// TIA Portal V21 export
FUNCTION "VACCUM" : Void   // FC12, LAD
{ S7_Optimized_Access := 'TRUE' }
// stored: SetENOAutomatically false
   VAR_TEMP
      "VACCUM DIFF" : Real;
      "VACCUM LEAK DIFF" : Real;
   END_VAR
   VAR_TEMP   // added for the SCL form of the ladder/FBD networks
      _w1 : Bool;
      _w2 : Bool;
      _w3 : Bool;
      _w4 : Bool;
      _w5 : Bool;
      _w6 : Bool;
      _w7 : Bool;
      _w8 : Bool;
      _w9 : Bool;
      _w10 : Bool;
      _w11 : Bool;
      _w12 : Bool;
      _w13 : Bool;
      _w14 : Bool;
      _w15 : Bool;
      _w16 : Bool;
      _w17 : Bool;
      _w18 : Bool;
      _w19 : Bool;
      _w20 : Bool;
   END_VAR
BEGIN

REGION Network 1
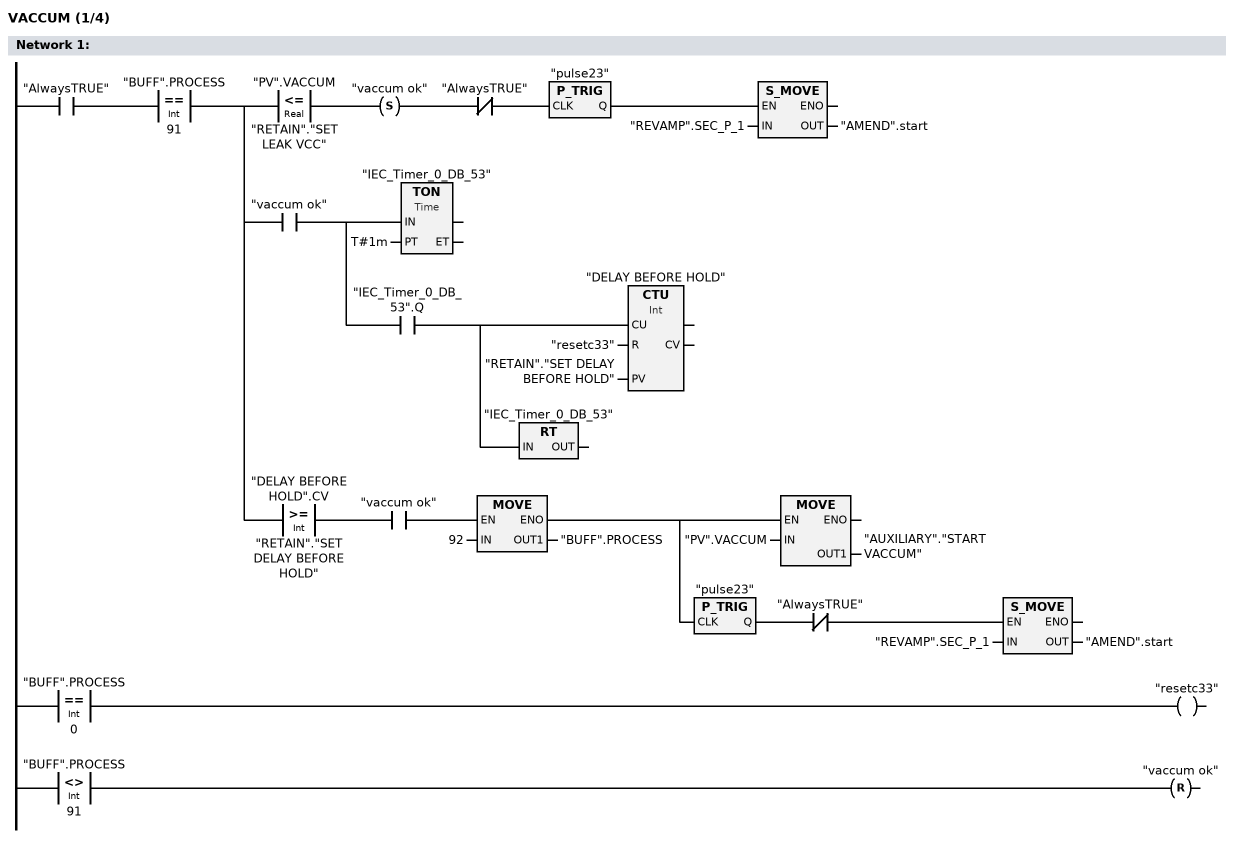
   RUNG wire#powerrail
      Contact( "AlwaysTRUE" )
      { S7_Templates := "SrcType := Int" } EQ_Contact(in1 := "BUFF".PROCESS, in2 := 91)
      wire#w1
      { S7_Templates := "SrcType := Real" } LE_Contact(in1 := "PV".VACCUM, in2 := "RETAIN"."SET LEAK VCC")
      S_Coil( "vaccum ok" )
      I_Contact( "AlwaysTRUE" )
      P_Trig( "pulse23" )
      S_Move(in := "REVAMP".SEC_P_1, out => "AMEND".start)
   END_RUNG
   RUNG wire#w1
      Contact( "vaccum ok" )
      wire#w2
      { S7_Templates := "time_type := Time" } "IEC_Timer_0_DB_53".TON(pt := T#1m, et =>)
   END_RUNG
   RUNG wire#w2
      Contact( "IEC_Timer_0_DB_53".Q )
      wire#w3
      { S7_Templates := "value_type := Int" } "DELAY BEFORE HOLD".CTU(r := "resetc33", pv := "RETAIN"."SET DELAY BEFORE HOLD", cv =>)
   END_RUNG
   RUNG wire#w3
      RT_Coil( "IEC_Timer_0_DB_53" )
   END_RUNG
   RUNG wire#w1
      { S7_Templates := "SrcType := Int" } GE_Contact(in1 := "DELAY BEFORE HOLD".CV, in2 := "RETAIN"."SET DELAY BEFORE HOLD")
      Contact( "vaccum ok" )
      Move(in := 92, out1 => "BUFF".PROCESS)
      wire#w4
      Move(in := "PV".VACCUM, out1 => "AUXILIARY"."START VACCUM")
   END_RUNG
   RUNG wire#w4
      P_Trig( "pulse23" )
      I_Contact( "AlwaysTRUE" )
      S_Move(in := "REVAMP".SEC_P_1, out => "AMEND".start)
   END_RUNG
   RUNG wire#powerrail
      { S7_Templates := "SrcType := Int" } EQ_Contact(in1 := "BUFF".PROCESS, in2 := 0)
      Coil( "resetc33" )
   END_RUNG
   RUNG wire#powerrail
      { S7_Templates := "SrcType := Int" } NE_Contact(in1 := "BUFF".PROCESS, in2 := 91)
      R_Coil( "vaccum ok" )
   END_RUNG
   // the same network as SCL:
   #_w1 := "AlwaysTRUE" AND ("BUFF".PROCESS = 91);
   #_w2 := #_w1 AND ("PV".VACCUM <= "RETAIN"."SET LEAK VCC");
   IF #_w2 THEN "vaccum ok" := TRUE; END_IF;
   #_w3 := #_w2 AND NOT "AlwaysTRUE";
   #_w4 := #_w3 AND NOT "pulse23";   // rising edge
   "pulse23" := #_w3;
   IF #_w4 THEN "AMEND".start := "REVAMP".SEC_P_1; END_IF;
   #_w5 := #_w1 AND "vaccum ok";
   "IEC_Timer_0_DB_53".TON(IN := #_w5, PT := T#1m);
   #_w6 := #_w5 AND "IEC_Timer_0_DB_53".Q;
   "DELAY BEFORE HOLD".CTU(CU := #_w6, R := "resetc33", PV := "RETAIN"."SET DELAY BEFORE HOLD");
   IF #_w6 THEN RESET_TIMER("IEC_Timer_0_DB_53"); END_IF;
   #_w7 := #_w1 AND ("DELAY BEFORE HOLD".CV >= "RETAIN"."SET DELAY BEFORE HOLD") AND "vaccum ok";
   IF #_w7 THEN
       "BUFF".PROCESS := 92;
       "AUXILIARY"."START VACCUM" := "PV".VACCUM;
   END_IF;
   #_w8 := #_w7 AND NOT "pulse23";   // rising edge
   "pulse23" := #_w7;
   IF #_w8 AND NOT "AlwaysTRUE" THEN "AMEND".start := "REVAMP".SEC_P_1; END_IF;
   "resetc33" := "BUFF".PROCESS = 0;
   IF "BUFF".PROCESS <> 91 THEN "vaccum ok" := FALSE; END_IF;
END_REGION

REGION Network 2
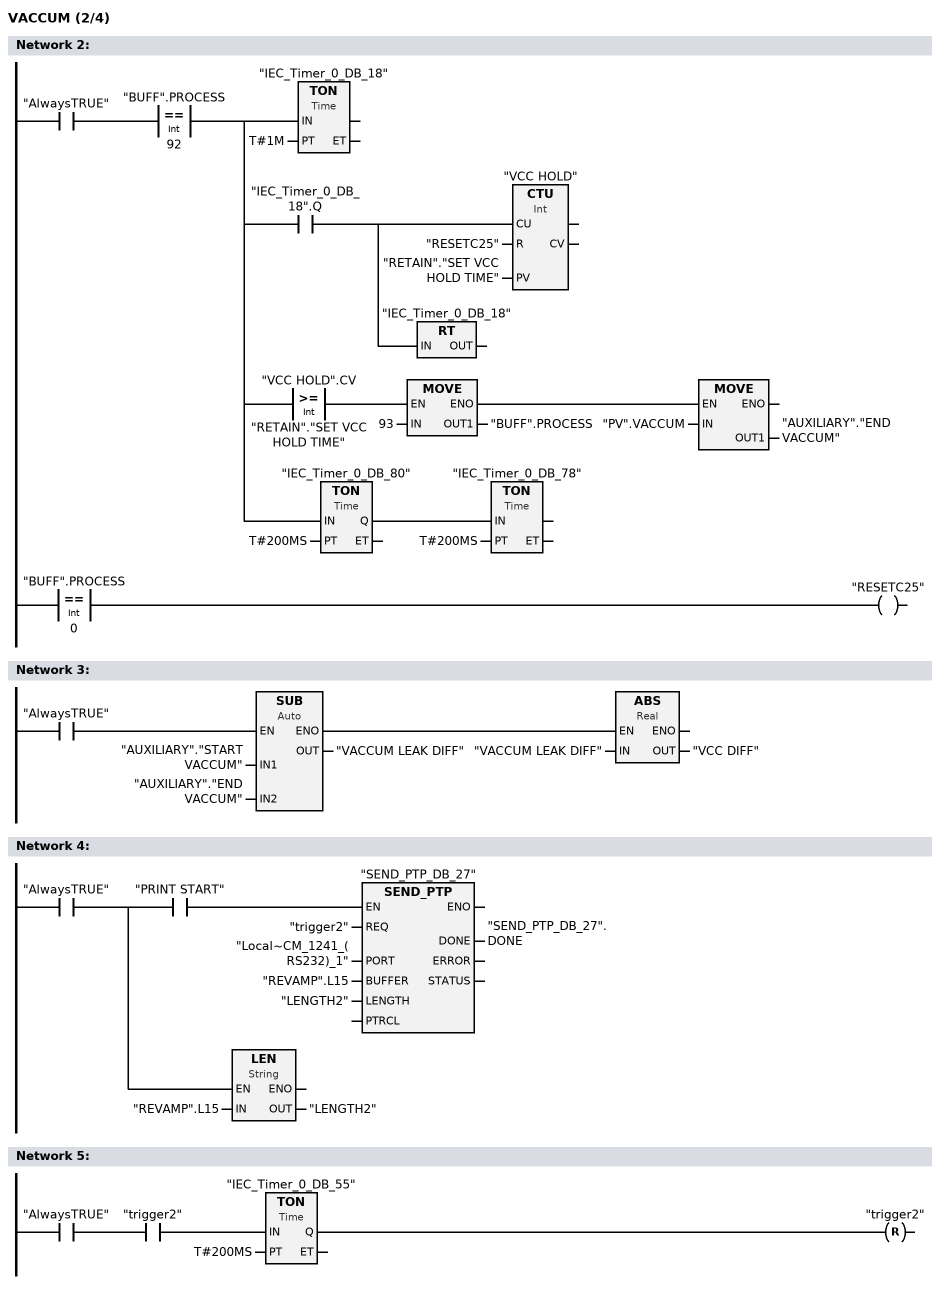
   RUNG wire#powerrail
      Contact( "AlwaysTRUE" )
      { S7_Templates := "SrcType := Int" } EQ_Contact(in1 := "BUFF".PROCESS, in2 := 92)
      wire#w1
      { S7_Templates := "time_type := Time" } "IEC_Timer_0_DB_18".TON(pt := T#1M, et =>)
   END_RUNG
   RUNG wire#w1
      Contact( "IEC_Timer_0_DB_18".Q )
      wire#w2
      { S7_Templates := "value_type := Int" } "VCC HOLD".CTU(r := "RESETC25", pv := "RETAIN"."SET VCC HOLD TIME", cv =>)
   END_RUNG
   RUNG wire#w2
      RT_Coil( "IEC_Timer_0_DB_18" )
   END_RUNG
   RUNG wire#w1
      { S7_Templates := "SrcType := Int" } GE_Contact(in1 := "VCC HOLD".CV, in2 := "RETAIN"."SET VCC HOLD TIME")
      Move(in := 93, out1 => "BUFF".PROCESS)
      Move(in := "PV".VACCUM, out1 => "AUXILIARY"."END VACCUM")
   END_RUNG
   RUNG wire#w1
      { S7_Templates := "time_type := Time" } "IEC_Timer_0_DB_80".TON(pt := T#200MS, et =>)
      { S7_Templates := "time_type := Time" } "IEC_Timer_0_DB_78".TON(pt := T#200MS, et =>)
   END_RUNG
   RUNG wire#powerrail
      { S7_Templates := "SrcType := Int" } EQ_Contact(in1 := "BUFF".PROCESS, in2 := 0)
      Coil( "RESETC25" )
   END_RUNG
   // the same network as SCL:
   #_w1 := "AlwaysTRUE" AND ("BUFF".PROCESS = 92);
   "IEC_Timer_0_DB_18".TON(IN := #_w1, PT := T#1M);
   #_w2 := #_w1 AND "IEC_Timer_0_DB_18".Q;
   "VCC HOLD".CTU(CU := #_w2, R := "RESETC25", PV := "RETAIN"."SET VCC HOLD TIME");
   IF #_w2 THEN RESET_TIMER("IEC_Timer_0_DB_18"); END_IF;
   IF #_w1 AND ("VCC HOLD".CV >= "RETAIN"."SET VCC HOLD TIME") THEN
       "BUFF".PROCESS := 93;
       "AUXILIARY"."END VACCUM" := "PV".VACCUM;
   END_IF;
   "IEC_Timer_0_DB_80".TON(IN := #_w1, PT := T#200MS);
   "IEC_Timer_0_DB_78".TON(IN := "IEC_Timer_0_DB_80".Q, PT := T#200MS);
   "RESETC25" := "BUFF".PROCESS = 0;
END_REGION

REGION Network 3
   RUNG wire#powerrail
      Contact( "AlwaysTRUE" )
      Sub(in1 := "AUXILIARY"."START VACCUM", in2 := "AUXILIARY"."END VACCUM", out => "VACCUM LEAK DIFF")
      { S7_Templates := "SrcType := Real" } Abs(in := "VACCUM LEAK DIFF", out => "VCC DIFF")
   END_RUNG
   // the same network as SCL:
   IF "AlwaysTRUE" THEN
       "VACCUM LEAK DIFF" := "AUXILIARY"."START VACCUM" - "AUXILIARY"."END VACCUM";
       "VCC DIFF" := ABS("VACCUM LEAK DIFF");
   END_IF;
END_REGION

REGION Network 4
   RUNG wire#powerrail
      Contact( "AlwaysTRUE" )
      wire#w1
      Contact( "PRINT START" )
      "SEND_PTP_DB_27".SEND_PTP(REQ := "trigger2", PORT := "Local~CM_1241_(RS232)_1", BUFFER := "REVAMP".L15, LENGTH := "LENGTH2", PTRCL :=, DONE => "SEND_PTP_DB_27".DONE, ERROR =>, STATUS =>)
   END_RUNG
   RUNG wire#w1
      { S7_Templates := "[str_type := String, return_type := Int]" } LEN(IN := "REVAMP".L15, OUT => "LENGTH2")
   END_RUNG
   // the same network as SCL:
   #_w1 := "AlwaysTRUE";
   IF "AlwaysTRUE" AND "PRINT START" THEN
       "SEND_PTP_DB_27"(REQ := "trigger2",   // SEND_PTP
                        PORT := "Local~CM_1241_(RS232)_1",
                        BUFFER := "REVAMP".L15,
                        LENGTH := "LENGTH2",
                        DONE => "SEND_PTP_DB_27".DONE);
   END_IF;
   IF #_w1 THEN LEN(IN := "REVAMP".L15, OUT => "LENGTH2"); END_IF;
END_REGION

REGION Network 5
   RUNG wire#powerrail
      Contact( "AlwaysTRUE" )
      Contact( "trigger2" )
      { S7_Templates := "time_type := Time" } "IEC_Timer_0_DB_55".TON(pt := T#200MS, et =>)
      R_Coil( "trigger2" )
   END_RUNG
   // the same network as SCL:
   "IEC_Timer_0_DB_55".TON(IN := "AlwaysTRUE" AND "trigger2", PT := T#200MS);
   IF "IEC_Timer_0_DB_55".Q THEN "trigger2" := FALSE; END_IF;
END_REGION

REGION Network 6
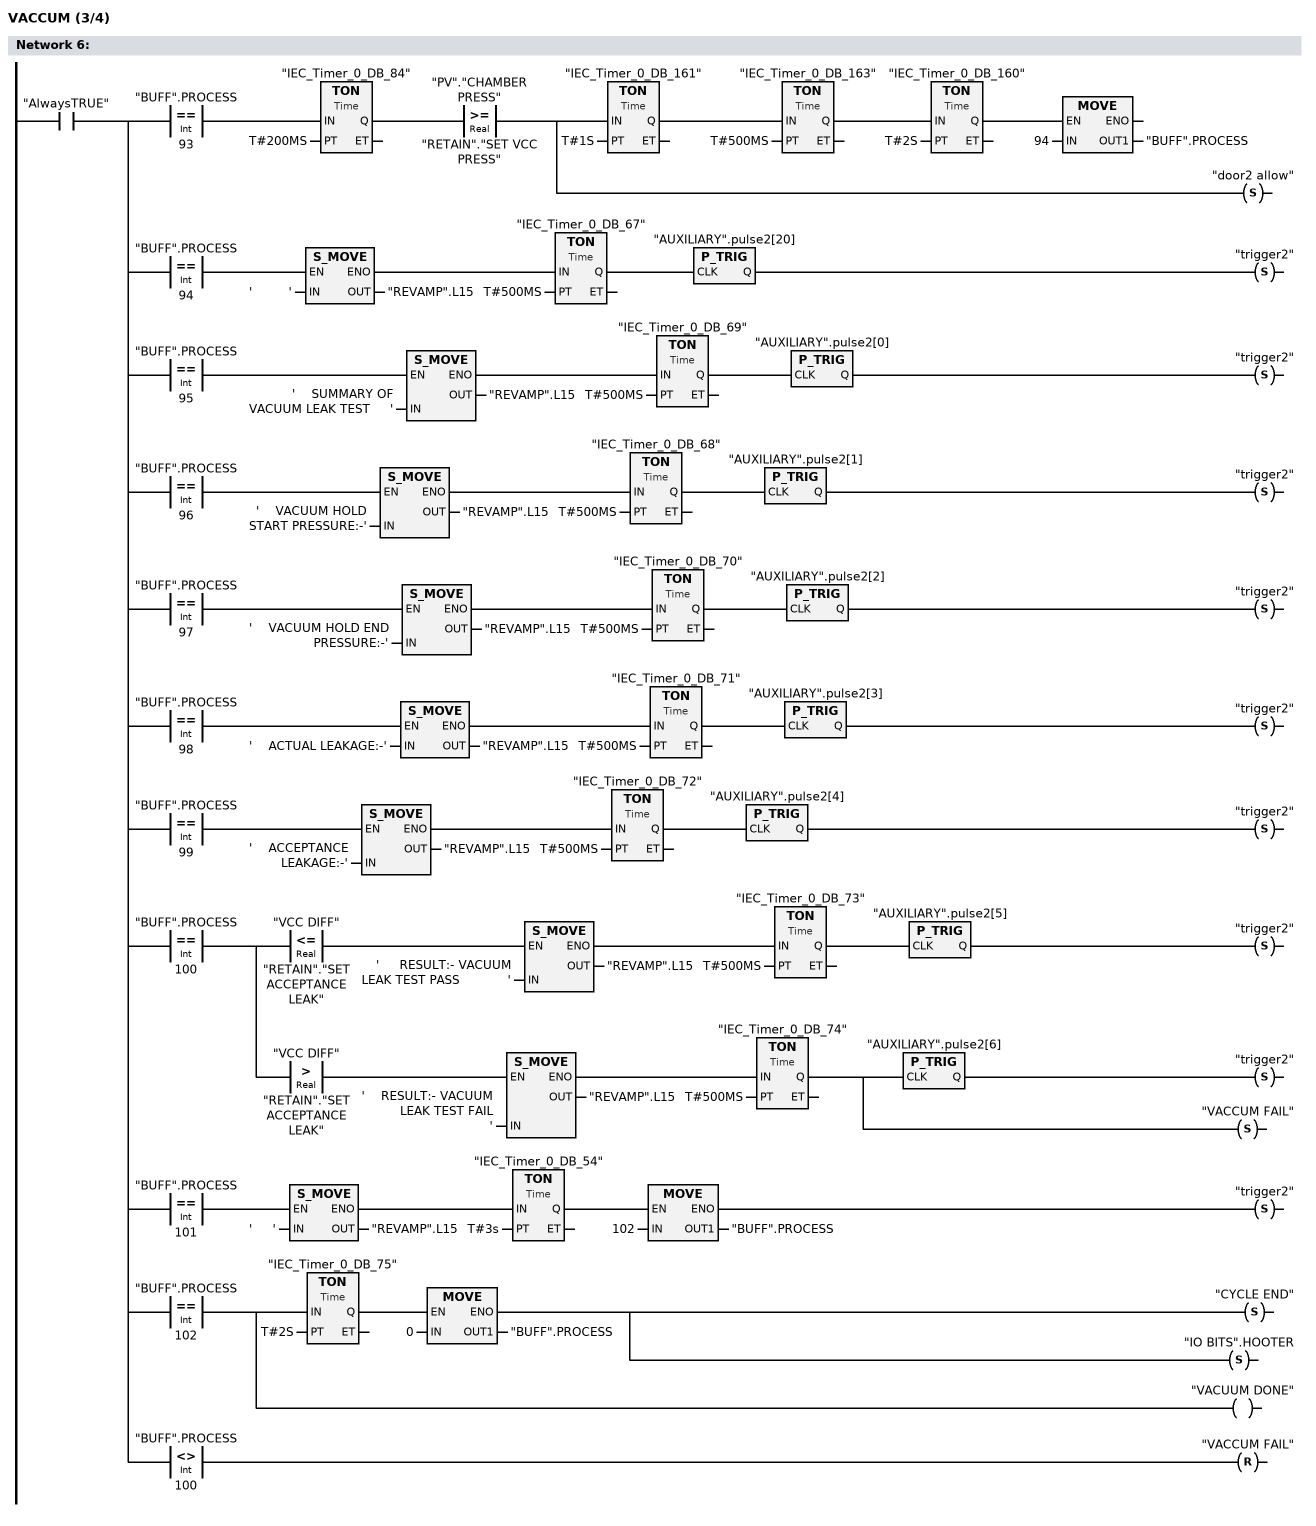
   RUNG wire#powerrail
      Contact( "AlwaysTRUE" )
      wire#w1
      { S7_Templates := "SrcType := Int" } EQ_Contact(in1 := "BUFF".PROCESS, in2 := 93)
      { S7_Templates := "time_type := Time" } "IEC_Timer_0_DB_84".TON(pt := T#200MS, et =>)
      { S7_Templates := "SrcType := Real" } GE_Contact(in1 := "PV"."CHAMBER PRESS", in2 := "RETAIN"."SET VCC PRESS")
      wire#w2
      { S7_Templates := "time_type := Time" } "IEC_Timer_0_DB_161".TON(pt := T#1S, et =>)
      { S7_Templates := "time_type := Time" } "IEC_Timer_0_DB_163".TON(pt := T#500MS, et =>)
      { S7_Templates := "time_type := Time" } "IEC_Timer_0_DB_160".TON(pt := T#2S, et =>)
      Move(in := 94, out1 => "BUFF".PROCESS)
   END_RUNG
   RUNG wire#w2
      S_Coil( "door2 allow" )
   END_RUNG
   RUNG wire#w1
      { S7_Templates := "SrcType := Int" } EQ_Contact(in1 := "BUFF".PROCESS, in2 := 94)
      S_Move(in := '         ', out => "REVAMP".L15)
      { S7_Templates := "time_type := Time" } "IEC_Timer_0_DB_67".TON(pt := T#500MS, et =>)
      P_Trig( "AUXILIARY".pulse2[20] )
      S_Coil( "trigger2" )
   END_RUNG
   RUNG wire#w1
      { S7_Templates := "SrcType := Int" } EQ_Contact(in1 := "BUFF".PROCESS, in2 := 95)
      S_Move(in := '    SUMMARY OF VACUUM LEAK TEST     ', out => "REVAMP".L15)
      { S7_Templates := "time_type := Time" } "IEC_Timer_0_DB_69".TON(pt := T#500MS, et =>)
      P_Trig( "AUXILIARY".pulse2[0] )
      S_Coil( "trigger2" )
   END_RUNG
   RUNG wire#w1
      { S7_Templates := "SrcType := Int" } EQ_Contact(in1 := "BUFF".PROCESS, in2 := 96)
      S_Move(in := '    VACUUM HOLD START PRESSURE:-', out => "REVAMP".L15)
      { S7_Templates := "time_type := Time" } "IEC_Timer_0_DB_68".TON(pt := T#500MS, et =>)
      P_Trig( "AUXILIARY".pulse2[1] )
      S_Coil( "trigger2" )
   END_RUNG
   RUNG wire#w1
      { S7_Templates := "SrcType := Int" } EQ_Contact(in1 := "BUFF".PROCESS, in2 := 97)
      S_Move(in := '    VACUUM HOLD END PRESSURE:-', out => "REVAMP".L15)
      { S7_Templates := "time_type := Time" } "IEC_Timer_0_DB_70".TON(pt := T#500MS, et =>)
      P_Trig( "AUXILIARY".pulse2[2] )
      S_Coil( "trigger2" )
   END_RUNG
   RUNG wire#w1
      { S7_Templates := "SrcType := Int" } EQ_Contact(in1 := "BUFF".PROCESS, in2 := 98)
      S_Move(in := '    ACTUAL LEAKAGE:-', out => "REVAMP".L15)
      { S7_Templates := "time_type := Time" } "IEC_Timer_0_DB_71".TON(pt := T#500MS, et =>)
      P_Trig( "AUXILIARY".pulse2[3] )
      S_Coil( "trigger2" )
   END_RUNG
   RUNG wire#w1
      { S7_Templates := "SrcType := Int" } EQ_Contact(in1 := "BUFF".PROCESS, in2 := 99)
      S_Move(in := '    ACCEPTANCE LEAKAGE:-', out => "REVAMP".L15)
      { S7_Templates := "time_type := Time" } "IEC_Timer_0_DB_72".TON(pt := T#500MS, et =>)
      P_Trig( "AUXILIARY".pulse2[4] )
      S_Coil( "trigger2" )
   END_RUNG
   RUNG wire#w1
      { S7_Templates := "SrcType := Int" } EQ_Contact(in1 := "BUFF".PROCESS, in2 := 100)
      wire#w3
      { S7_Templates := "SrcType := Real" } LE_Contact(in1 := "VCC DIFF", in2 := "RETAIN"."SET ACCEPTANCE LEAK")
      S_Move(in := '     RESULT:- VACUUM LEAK TEST PASS            ', out => "REVAMP".L15)
      { S7_Templates := "time_type := Time" } "IEC_Timer_0_DB_73".TON(pt := T#500MS, et =>)
      P_Trig( "AUXILIARY".pulse2[5] )
      S_Coil( "trigger2" )
   END_RUNG
   RUNG wire#w3
      { S7_Templates := "SrcType := Real" } GT_Contact(in1 := "VCC DIFF", in2 := "RETAIN"."SET ACCEPTANCE LEAK")
      S_Move(in := '    RESULT:- VACUUM LEAK TEST FAIL                   ', out => "REVAMP".L15)
      { S7_Templates := "time_type := Time" } "IEC_Timer_0_DB_74".TON(pt := T#500MS, et =>)
      wire#w4
      P_Trig( "AUXILIARY".pulse2[6] )
      S_Coil( "trigger2" )
   END_RUNG
   RUNG wire#w4
      S_Coil( "VACCUM FAIL" )
   END_RUNG
   RUNG wire#w1
      { S7_Templates := "SrcType := Int" } EQ_Contact(in1 := "BUFF".PROCESS, in2 := 101)
      S_Move(in := '     ', out => "REVAMP".L15)
      { S7_Templates := "time_type := Time" } "IEC_Timer_0_DB_54".TON(pt := T#3s, et =>)
      Move(in := 102, out1 => "BUFF".PROCESS)
      S_Coil( "trigger2" )
   END_RUNG
   RUNG wire#w1
      { S7_Templates := "SrcType := Int" } EQ_Contact(in1 := "BUFF".PROCESS, in2 := 102)
      wire#w5
      { S7_Templates := "time_type := Time" } "IEC_Timer_0_DB_75".TON(pt := T#2S, et =>)
      Move(in := 0, out1 => "BUFF".PROCESS)
      wire#w6
      S_Coil( "CYCLE END" )
   END_RUNG
   RUNG wire#w6
      S_Coil( "IO BITS".HOOTER )
   END_RUNG
   RUNG wire#w5
      Coil( "VACUUM DONE" )
   END_RUNG
   RUNG wire#w1
      { S7_Templates := "SrcType := Int" } NE_Contact(in1 := "BUFF".PROCESS, in2 := 100)
      R_Coil( "VACCUM FAIL" )
   END_RUNG
   // the same network as SCL:
   "IEC_Timer_0_DB_84".TON(IN := "AlwaysTRUE" AND ("BUFF".PROCESS = 93), PT := T#200MS);
   #_w1 := "IEC_Timer_0_DB_84".Q AND ("PV"."CHAMBER PRESS" >= "RETAIN"."SET VCC PRESS");
   "IEC_Timer_0_DB_161".TON(IN := #_w1, PT := T#1S);
   "IEC_Timer_0_DB_163".TON(IN := "IEC_Timer_0_DB_161".Q, PT := T#500MS);
   "IEC_Timer_0_DB_160".TON(IN := "IEC_Timer_0_DB_163".Q, PT := T#2S);
   IF "IEC_Timer_0_DB_160".Q THEN "BUFF".PROCESS := 94; END_IF;
   IF #_w1 THEN "door2 allow" := TRUE; END_IF;
   #_w2 := "AlwaysTRUE" AND ("BUFF".PROCESS = 94);
   IF #_w2 THEN "REVAMP".L15 := '         '; END_IF;
   "IEC_Timer_0_DB_67".TON(IN := #_w2, PT := T#500MS);
   #_w3 := "IEC_Timer_0_DB_67".Q AND NOT "AUXILIARY".pulse2[20];   // rising edge
   "AUXILIARY".pulse2[20] := "IEC_Timer_0_DB_67".Q;
   IF #_w3 THEN "trigger2" := TRUE; END_IF;
   #_w4 := "AlwaysTRUE" AND ("BUFF".PROCESS = 95);
   IF #_w4 THEN "REVAMP".L15 := '    SUMMARY OF VACUUM LEAK TEST     '; END_IF;
   "IEC_Timer_0_DB_69".TON(IN := #_w4, PT := T#500MS);
   #_w5 := "IEC_Timer_0_DB_69".Q AND NOT "AUXILIARY".pulse2[0];   // rising edge
   "AUXILIARY".pulse2[0] := "IEC_Timer_0_DB_69".Q;
   IF #_w5 THEN "trigger2" := TRUE; END_IF;
   #_w6 := "AlwaysTRUE" AND ("BUFF".PROCESS = 96);
   IF #_w6 THEN "REVAMP".L15 := '    VACUUM HOLD START PRESSURE:-'; END_IF;
   "IEC_Timer_0_DB_68".TON(IN := #_w6, PT := T#500MS);
   #_w7 := "IEC_Timer_0_DB_68".Q AND NOT "AUXILIARY".pulse2[1];   // rising edge
   "AUXILIARY".pulse2[1] := "IEC_Timer_0_DB_68".Q;
   IF #_w7 THEN "trigger2" := TRUE; END_IF;
   #_w8 := "AlwaysTRUE" AND ("BUFF".PROCESS = 97);
   IF #_w8 THEN "REVAMP".L15 := '    VACUUM HOLD END PRESSURE:-'; END_IF;
   "IEC_Timer_0_DB_70".TON(IN := #_w8, PT := T#500MS);
   #_w9 := "IEC_Timer_0_DB_70".Q AND NOT "AUXILIARY".pulse2[2];   // rising edge
   "AUXILIARY".pulse2[2] := "IEC_Timer_0_DB_70".Q;
   IF #_w9 THEN "trigger2" := TRUE; END_IF;
   #_w10 := "AlwaysTRUE" AND ("BUFF".PROCESS = 98);
   IF #_w10 THEN "REVAMP".L15 := '    ACTUAL LEAKAGE:-'; END_IF;
   "IEC_Timer_0_DB_71".TON(IN := #_w10, PT := T#500MS);
   #_w11 := "IEC_Timer_0_DB_71".Q AND NOT "AUXILIARY".pulse2[3];   // rising edge
   "AUXILIARY".pulse2[3] := "IEC_Timer_0_DB_71".Q;
   IF #_w11 THEN "trigger2" := TRUE; END_IF;
   #_w12 := "AlwaysTRUE" AND ("BUFF".PROCESS = 99);
   IF #_w12 THEN "REVAMP".L15 := '    ACCEPTANCE LEAKAGE:-'; END_IF;
   "IEC_Timer_0_DB_72".TON(IN := #_w12, PT := T#500MS);
   #_w13 := "IEC_Timer_0_DB_72".Q AND NOT "AUXILIARY".pulse2[4];   // rising edge
   "AUXILIARY".pulse2[4] := "IEC_Timer_0_DB_72".Q;
   IF #_w13 THEN "trigger2" := TRUE; END_IF;
   #_w14 := "AlwaysTRUE" AND ("BUFF".PROCESS = 100);
   #_w15 := #_w14 AND ("VCC DIFF" <= "RETAIN"."SET ACCEPTANCE LEAK");
   IF #_w15 THEN "REVAMP".L15 := '     RESULT:- VACUUM LEAK TEST PASS            '; END_IF;
   "IEC_Timer_0_DB_73".TON(IN := #_w15, PT := T#500MS);
   #_w16 := "IEC_Timer_0_DB_73".Q AND NOT "AUXILIARY".pulse2[5];   // rising edge
   "AUXILIARY".pulse2[5] := "IEC_Timer_0_DB_73".Q;
   IF #_w16 THEN "trigger2" := TRUE; END_IF;
   #_w17 := #_w14 AND ("VCC DIFF" > "RETAIN"."SET ACCEPTANCE LEAK");
   IF #_w17 THEN "REVAMP".L15 := '    RESULT:- VACUUM LEAK TEST FAIL                   '; END_IF;
   "IEC_Timer_0_DB_74".TON(IN := #_w17, PT := T#500MS);
   #_w18 := "IEC_Timer_0_DB_74".Q AND NOT "AUXILIARY".pulse2[6];   // rising edge
   "AUXILIARY".pulse2[6] := "IEC_Timer_0_DB_74".Q;
   IF #_w18 THEN "trigger2" := TRUE; END_IF;
   IF "IEC_Timer_0_DB_74".Q THEN "VACCUM FAIL" := TRUE; END_IF;
   #_w19 := "AlwaysTRUE" AND ("BUFF".PROCESS = 101);
   IF #_w19 THEN "REVAMP".L15 := '     '; END_IF;
   "IEC_Timer_0_DB_54".TON(IN := #_w19, PT := T#3s);
   IF "IEC_Timer_0_DB_54".Q THEN
       "BUFF".PROCESS := 102;
       "trigger2" := TRUE;
   END_IF;
   #_w20 := "AlwaysTRUE" AND ("BUFF".PROCESS = 102);
   "IEC_Timer_0_DB_75".TON(IN := #_w20, PT := T#2S);
   IF "IEC_Timer_0_DB_75".Q THEN
       "BUFF".PROCESS := 0;
       "CYCLE END" := TRUE;
       "IO BITS".HOOTER := TRUE;
   END_IF;
   "VACUUM DONE" := #_w20;
   IF "AlwaysTRUE" AND ("BUFF".PROCESS <> 100) THEN "VACCUM FAIL" := FALSE; END_IF;
END_REGION

REGION Network 7
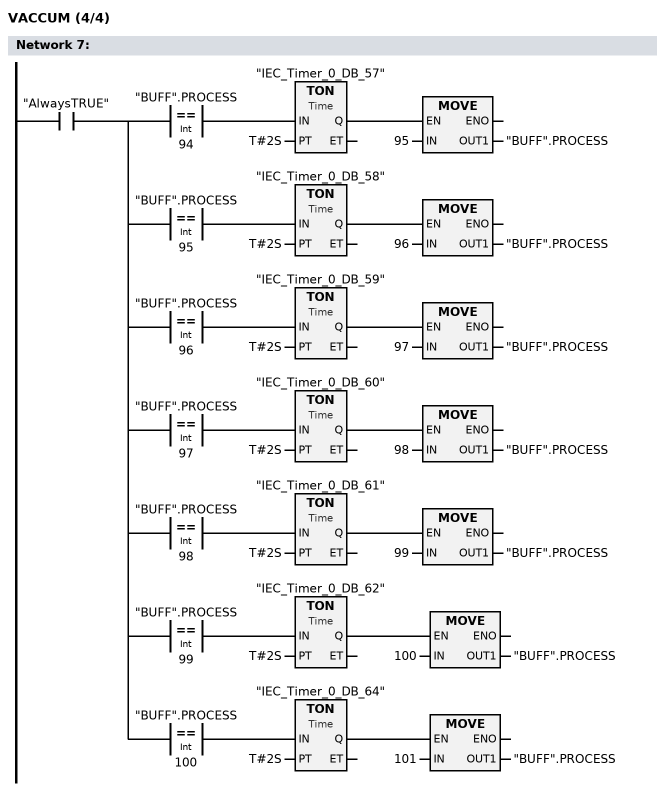
   RUNG wire#powerrail
      Contact( "AlwaysTRUE" )
      wire#w1
      { S7_Templates := "SrcType := Int" } EQ_Contact(in1 := "BUFF".PROCESS, in2 := 94)
      { S7_Templates := "time_type := Time" } "IEC_Timer_0_DB_57".TON(pt := T#2S, et =>)
      Move(in := 95, out1 => "BUFF".PROCESS)
   END_RUNG
   RUNG wire#w1
      { S7_Templates := "SrcType := Int" } EQ_Contact(in1 := "BUFF".PROCESS, in2 := 95)
      { S7_Templates := "time_type := Time" } "IEC_Timer_0_DB_58".TON(pt := T#2S, et =>)
      Move(in := 96, out1 => "BUFF".PROCESS)
   END_RUNG
   RUNG wire#w1
      { S7_Templates := "SrcType := Int" } EQ_Contact(in1 := "BUFF".PROCESS, in2 := 96)
      { S7_Templates := "time_type := Time" } "IEC_Timer_0_DB_59".TON(pt := T#2S, et =>)
      Move(in := 97, out1 => "BUFF".PROCESS)
   END_RUNG
   RUNG wire#w1
      { S7_Templates := "SrcType := Int" } EQ_Contact(in1 := "BUFF".PROCESS, in2 := 97)
      { S7_Templates := "time_type := Time" } "IEC_Timer_0_DB_60".TON(pt := T#2S, et =>)
      Move(in := 98, out1 => "BUFF".PROCESS)
   END_RUNG
   RUNG wire#w1
      { S7_Templates := "SrcType := Int" } EQ_Contact(in1 := "BUFF".PROCESS, in2 := 98)
      { S7_Templates := "time_type := Time" } "IEC_Timer_0_DB_61".TON(pt := T#2S, et =>)
      Move(in := 99, out1 => "BUFF".PROCESS)
   END_RUNG
   RUNG wire#w1
      { S7_Templates := "SrcType := Int" } EQ_Contact(in1 := "BUFF".PROCESS, in2 := 99)
      { S7_Templates := "time_type := Time" } "IEC_Timer_0_DB_62".TON(pt := T#2S, et =>)
      Move(in := 100, out1 => "BUFF".PROCESS)
   END_RUNG
   RUNG wire#w1
      { S7_Templates := "SrcType := Int" } EQ_Contact(in1 := "BUFF".PROCESS, in2 := 100)
      { S7_Templates := "time_type := Time" } "IEC_Timer_0_DB_64".TON(pt := T#2S, et =>)
      Move(in := 101, out1 => "BUFF".PROCESS)
   END_RUNG
   // the same network as SCL:
   "IEC_Timer_0_DB_57".TON(IN := "AlwaysTRUE" AND ("BUFF".PROCESS = 94), PT := T#2S);
   IF "IEC_Timer_0_DB_57".Q THEN "BUFF".PROCESS := 95; END_IF;
   "IEC_Timer_0_DB_58".TON(IN := "AlwaysTRUE" AND ("BUFF".PROCESS = 95), PT := T#2S);
   IF "IEC_Timer_0_DB_58".Q THEN "BUFF".PROCESS := 96; END_IF;
   "IEC_Timer_0_DB_59".TON(IN := "AlwaysTRUE" AND ("BUFF".PROCESS = 96), PT := T#2S);
   IF "IEC_Timer_0_DB_59".Q THEN "BUFF".PROCESS := 97; END_IF;
   "IEC_Timer_0_DB_60".TON(IN := "AlwaysTRUE" AND ("BUFF".PROCESS = 97), PT := T#2S);
   IF "IEC_Timer_0_DB_60".Q THEN "BUFF".PROCESS := 98; END_IF;
   "IEC_Timer_0_DB_61".TON(IN := "AlwaysTRUE" AND ("BUFF".PROCESS = 98), PT := T#2S);
   IF "IEC_Timer_0_DB_61".Q THEN "BUFF".PROCESS := 99; END_IF;
   "IEC_Timer_0_DB_62".TON(IN := "AlwaysTRUE" AND ("BUFF".PROCESS = 99), PT := T#2S);
   IF "IEC_Timer_0_DB_62".Q THEN "BUFF".PROCESS := 100; END_IF;
   "IEC_Timer_0_DB_64".TON(IN := "AlwaysTRUE" AND ("BUFF".PROCESS = 100), PT := T#2S);
   IF "IEC_Timer_0_DB_64".Q THEN "BUFF".PROCESS := 101; END_IF;
END_REGION
END_FUNCTION
